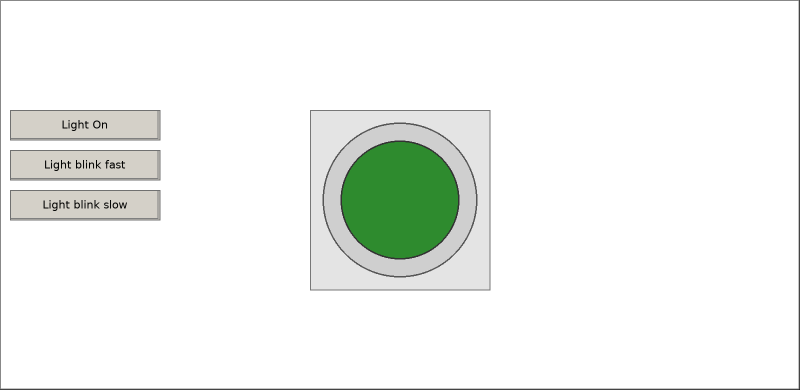
VISUALIZATION VisuPushbuttonLightControl  // 800x390
    Rectangle (0,0 800x390)
    PushSwitch (310,110 180x180), variable: GVL_DevManual.fbManualControler.pDevPBL^.bFcoInputActive, behaviour: TOGGLE, style: Switch-PushSwitch-Green
    Button (10,110 150x30), "Light On"
        toggle GVL_DevManual.fbManualControler.pDevPBL^.fbLight.bCmdOn
    Button (10,150 150x30), "Light blink fast"
        toggle GVL_DevManual.fbManualControler.pDevPBL^.fbLight.bCmdBlinkFast
    Button (10,190 150x30), "Light blink slow"
        toggle GVL_DevManual.fbManualControler.pDevPBL^.fbLight.bCmdBlinkSlow
END_VISUALIZATION

(* stored: Version 1.1.0.1, ProductVersion 3.1.4024.5
   Visu VisuPushbuttonLightControl: Id {b1000dcd-1831-44d9-b5dd-79a42998adcb} *)
